{attribute 'GeneratedUsingTerminal: EL6201-0000-0017'}
{attribute addProperty BoxType "EL6201-0000-0017"}
{attribute addProperty Id "Slave_21A_DI0BOOL1Slave_21A_DI1BOOL1Slave_21A_DI2BOOL1Slave_21A_DI3BOOL1Slave_21B_DI0BOOL1Slave_21B_DI1BOOL1Slave_21B_DI2BOOL1Slave_21B_DI3BOOL1"}
{attribute addProperty CRC "1146310512"}
{attribute addProperty Size "8"}
TYPE Slave_21_Inputs_44534F70 :
STRUCT
	{attribute addProperty Name "Slave_21A_DI0"}
	Slave_21A_DI0 : BOOL;
	{attribute addProperty Name "Slave_21A_DI1"}
	Slave_21A_DI1 : BOOL;
	{attribute addProperty Name "Slave_21A_DI2"}
	Slave_21A_DI2 : BOOL;
	{attribute addProperty Name "Slave_21A_DI3"}
	Slave_21A_DI3 : BOOL;
	{attribute addProperty Name "Slave_21B_DI0"}
	Slave_21B_DI0 : BOOL;
	{attribute addProperty Name "Slave_21B_DI1"}
	Slave_21B_DI1 : BOOL;
	{attribute addProperty Name "Slave_21B_DI2"}
	Slave_21B_DI2 : BOOL;
	{attribute addProperty Name "Slave_21B_DI3"}
	Slave_21B_DI3 : BOOL;
END_STRUCT
END_TYPE

(* stored: Version 1.2.0.0, ProductVersion 3.1.4024.9
   DUT Slave_21_Inputs_44534F70: Id {dbe39f1d-3df4-4e12-8dc3-6ef8476df124} *)
